// LS Electric XG5000 project: 16-42-1
// PLC NewPLC
// module base 0 slot 0: 입출력 모듈:XBC-DR14E (DC 24V 입력 8점, 릴레이 출력 6점)

PROGRAM NewProgram (task: 스캔 프로그램)

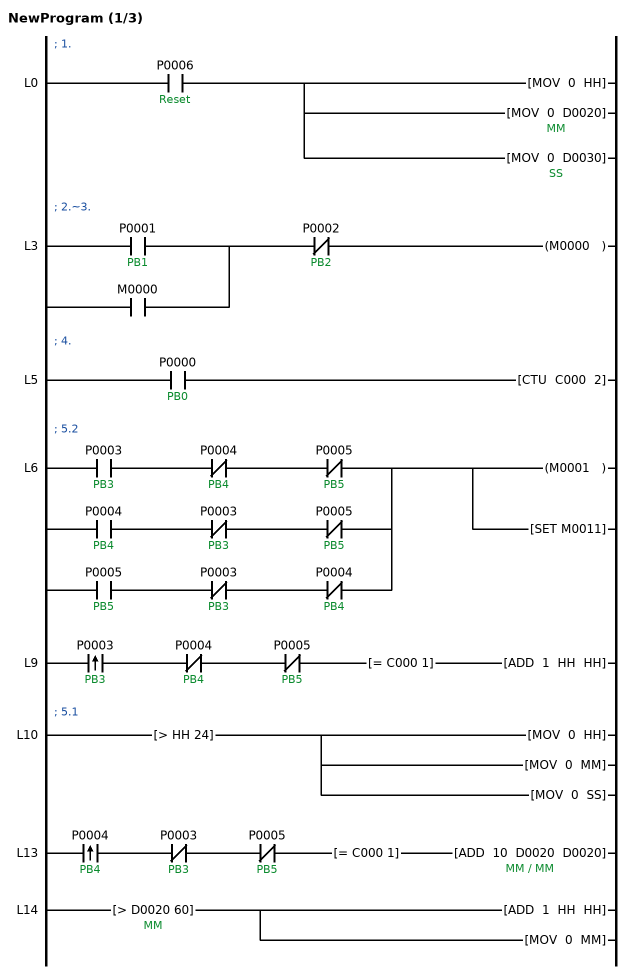
; L0
LOAD      P0006	// Reset
MOV       0 HH
MOV       0 D0020	// MM
MOV       0 D0030	// SS
// output comment: 1.
; L3
LOAD      P0001	// PB1
OR        M0000
AND NOT   P0002	// PB2
OUT       M0000
// output comment: 2.~3.
; L5
LOAD      P0000	// PB0
CTU       C000 2
// output comment: 4.
; L6
LOAD      P0003	// PB3
AND NOT   P0004	// PB4
AND NOT   P0005	// PB5
LOAD      P0004	// PB4
AND NOT   P0003	// PB3
AND NOT   P0005	// PB5
OR LOAD
LOAD      P0005	// PB5
AND NOT   P0003	// PB3
AND NOT   P0004	// PB4
OR LOAD
OUT       M0001
SET       M0011
// output comment: 5.2
; L9
LOADP     P0003	// PB3
AND NOT   P0004	// PB4
AND NOT   P0005	// PB5
AND=      C000 1
ADD       1 HH HH
; L10
LOAD>     HH 24
MOV       0 HH
MOV       0 MM
MOV       0 SS
// output comment: 5.1
; L13
LOADP     P0004	// PB4
AND NOT   P0003	// PB3
AND NOT   P0005	// PB5
AND=      C000 1
ADD       10 D0020 D0020	// MM / MM
; L14
LOAD>     D0020 60	// MM
ADD       1 HH HH
MOV       0 MM

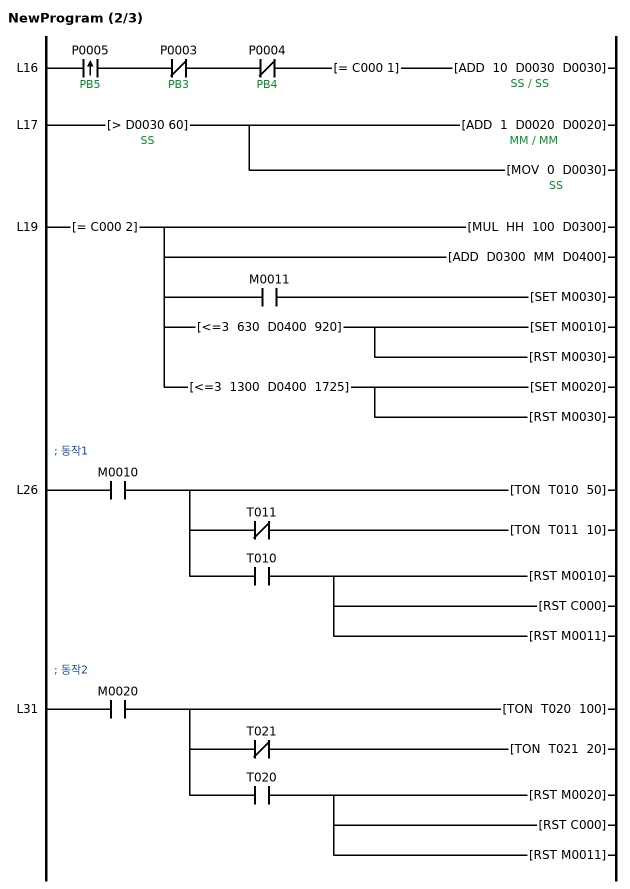
; L16
LOADP     P0005	// PB5
AND NOT   P0003	// PB3
AND NOT   P0004	// PB4
AND=      C000 1
ADD       10 D0030 D0030	// SS / SS
; L17
LOAD>     D0030 60	// SS
ADD       1 D0020 D0020	// MM / MM
MOV       0 D0030	// SS
; L19
LOAD=     C000 2
MUL       HH 100 D0300
ADD       D0300 MM D0400
MPUSH
AND       M0011
SET       M0030
MLOAD
AND<=3    630 D0400 920
SET       M0010
RST       M0030
MPOP
AND<=3    1300 D0400 1725
SET       M0020
RST       M0030
; L26
LOAD      M0010
TON       T010 50
MPUSH
AND NOT   T011
TON       T011 10
MPOP
AND       T010
RST       M0010
RST       C000
RST       M0011
// output comment: 동작1
; L31
LOAD      M0020
TON       T020 100
MPUSH
AND NOT   T021
TON       T021 20
MPOP
AND       T020
RST       M0020
RST       C000
RST       M0011
// output comment: 동작2

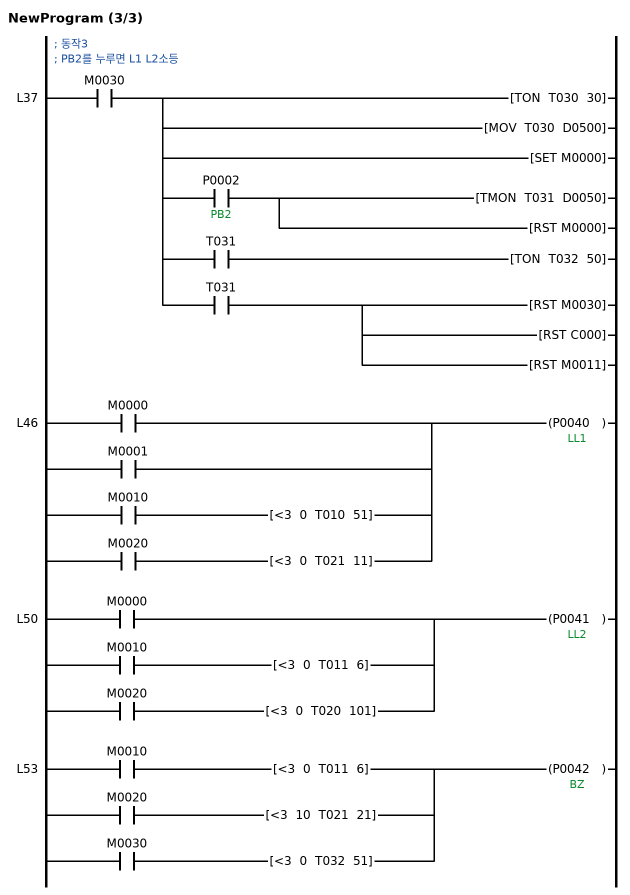
; L37
LOAD      M0030
TON       T030 30
MOV       T030 D0500
SET       M0000
MPUSH
AND       P0002	// PB2
TMON      T031 D0050
RST       M0000
MLOAD
AND       T031
TON       T032 50
MPOP
AND       T031
RST       M0030
RST       C000
RST       M0011
// output comment: 동작3
// output comment: PB2를 누루면 L1 L2소등
; L46
LOAD      M0000
OR        M0001
LOAD      M0010
AND<3     0 T010 51
OR LOAD
LOAD      M0020
AND<3     0 T021 11
OR LOAD
OUT       P0040	// LL1
; L50
LOAD      M0000
LOAD      M0010
AND<3     0 T011 6
OR LOAD
LOAD      M0020
AND<3     0 T020 101
OR LOAD
OUT       P0041	// LL2
; L53
LOAD      M0010
AND<3     0 T011 6
LOAD      M0020
AND<3     10 T021 21
OR LOAD
LOAD      M0030
AND<3     0 T032 51
OR LOAD
OUT       P0042	// BZ

VARIABLES AND COMMENTS (devices not used above)
D00010	WORD	HH